FUNCTION F_TimeNow : STRING
VAR_INPUT
END_VAR
VAR
	
END_VAR


//F_TimeNow := (GVL_General.DateTimeNow)

END_FUNCTION

(* stored: Version 1.1.0.1, ProductVersion 3.1.4022.16
   POU F_TimeNow: Id {d6d3adc2-e4a1-4220-80b1-5e9ccf54fff1}, SpecialFunc None *)
